{attribute 'pack_mode' := '0'}
TYPE ACMethodMixingR EXTENDS ACMethodBaseR :
STRUCT
	// Dauer 
	_ActDuration : TIME;
	//Temperatur
	_ActTemperature : LREAL;
END_STRUCT
END_TYPE

(* stored: Version 1.1.0.1, ProductVersion 3.1.4020.12
   DUT ACMethodMixingR: Id {473df5d3-5f72-4e00-8e52-1893886acc90} *)
